(* IEC 61131-3 sources: SRCI/RobotLibrary/RobotLibrary/POUs/_internal, 7 files *)

(* ---- ActiveCommandRegisterFB.st ---- *)
FUNCTION_BLOCK ActiveCommandRegisterFB EXTENDS RobotLibraryLogFB
// -------------------------------------------------------------------------
//  SRCI Robot Library
// -------------------------------------------------------------------------
//
//  Object:      ActiveCommandRegisterFB
//  Author:      Thorsten Brach
//  Date:        2024-06-01
//
//  Description:
//
//
//  Copyright:
//    (C) 2024 Thorsten Brach. All rights reserved
//             Licensed under the LGPL-3.0 license.
//
//  Disclaimer:
//    This project is provided without any guarantee and can be used for
//    private and commercial purposes. Any use is at the user’s
//    own risk and responsibility.
//
// -------------------------------------------------------------------------
VAR_INPUT
  /// Active Command Register
  Register            : ARRAY [1..RobotLibraryParameter.ACTIVE_CMD_REGISTER_ENTRIES_MAX] OF AxesGroupAcyclicAcrEntry;
  /// System Time
  SystemTime          : DT;
END_VAR

VAR_OUTPUT
  /// Size of the register
  Size                : UINT := DINT_TO_UINT(RobotLibraryParameter.ACTIVE_CMD_REGISTER_ENTRIES_MAX);
  /// Execution Order List
  ExecutionOrderList  : ARRAY [1..RobotLibraryParameter.ACTIVE_CMD_REGISTER_ENTRIES_MAX] OF DINT;
END_VAR

VAR
  /// temporarty Active Command Register
  TmpRegister        : ARRAY [1..RobotLibraryParameter.ACTIVE_CMD_REGISTER_ENTRIES_MAX] OF AxesGroupAcyclicAcrEntry;
  /// last used unique ID
  LastUniqueID       : UINT;
  ///

END_VAR

VAR CONSTANT
  /// Active command
  ACTIVE_CMD           : UDINT := 1;
  /// Buffered command
  BUFFER_CMD           : UDINT := 2;
  /// Empty ARC entry
  EMPTY_ARC_ENTRY      : AxesGroupAcyclicAcrEntry;
  /// Empty command entry
  EMPTY_CMD_ENTRY      : AxesGroupAcyclicAcrEntryCmdBuffer;

  /// constant for byte index of priority in payload
  PRIORITY_IDX         : BYTE := 3;  /// bitmask to mask the priority out of the halfbyte
  PRIORITY_BIT_MASK    : BYTE := 2#000_1111;
END_VAR

  ManageRegister();

  UpdateExecutionOrderList();

END_FUNCTION_BLOCK

METHOD PUBLIC AddCmd : UDINT
VAR_INPUT
  /// Pointer to the corresponding command-FB to enable a callback mechanism
  pCommandFB   : POINTER TO RobotLibraryBaseFB;
END_VAR

VAR
  /// internal index for loops
 _regIdx     : DINT;
  /// internal command type
 _cmdType    : CmdType;
  /// log message
 _messageLog         : AlarmMessage;
END_VAR

  FOR _regIdx := 1 TO RobotLibraryParameter.ACTIVE_CMD_REGISTER_ENTRIES_MAX
  DO
    IF ( Register[_regIdx].State = ActiveCommandRegisterState.IS_FREE )
    THEN
      Register[_regIdx].State                        := ActiveCommandRegisterState.IS_PROCESSING;
      Register[_regIdx].UniqueID                     := CreateUniqueID();
      Register[_regIdx].pCommandFB                   := pCommandFB;

      // check pointer to command FB
      IF ( Register[_regIdx].pCommandFB <> RobotLibraryConstants.XNULL )
      THEN
        Register[_regIdx].Command[RobotLibraryConstants.ACTIVE_CMD].Timestamp  := SystemTime;
        Register[_regIdx].Command[RobotLibraryConstants.ACTIVE_CMD].Payload    := pCommandFB^.CommandData.Payload;
        Register[_regIdx].Command[RobotLibraryConstants.ACTIVE_CMD].PayloadLen := pCommandFB^.CommandData.PayloadLen;
        Register[_regIdx].Command[RobotLibraryConstants.ACTIVE_CMD].PayLoadPtr := 0;
        Register[_regIdx].Command[RobotLibraryConstants.ACTIVE_CMD].State      := BufferStateCmd.CREATED;
  		END_IF

      // return Unique ID
      AddCmd := Register[_regIdx].UniqueID;

      // Get CmdType from payload
      MemCpy( destAddr := ADR(_cmdType), ADR(pCommandFB^.CommandData.Payload), SIZEOF(_cmdType));

      // Create log entry
      CreateLogMessagePara1 ( Timestamp   := SystemTime,
                              MessageType := MessageType.CMD,
                              Severity    := Severity.DEBUG,
                              MessageCode := 0,
                              MessageText := 'Added Cmd <{1}> to active command register',
                              Para1       :=  CmdTypeToString(SwapUint(_cmdType)));
      EXIT;
  	END_IF
  END_FOR

END_METHOD

METHOD AddRsp : UDINT
VAR_INPUT
  /// Response
  Rsp : TelegramRobToPlcFragment;
END_VAR
VAR
  /// internal index for loops
 _Idx             : DINT;
  /// internal registen index
 _regIdx          : DINT;
  /// internal FragmentAction
 _fragmentAction  :  FragmentAction;
  /// internal command message state
 _cmdMessageState : CmdMessageState;
END_VAR

  FOR _regIdx := 1 TO RobotLibraryParameter.ACTIVE_CMD_REGISTER_ENTRIES_MAX
  DO
    IF ( Register[_regIdx].UniqueID = Rsp.Header.CmdID )
    THEN
      // convert to fragment action
     _fragmentAction := ByteToFragmentAction(Rsp.Header.FragmentAction);

      // delete response
      IF ( _fragmentAction.Clear )
      THEN
        MemSet( ADR(Register[_regIdx].Response[1]), 0, SIZEOF(Register[_regIdx].Response[1]));
      END_IF

      // add payload to response
      FOR _idx := Rsp.Header.PayloadPointer TO  Rsp.Header.PayloadLength -1
      DO
        Register[_regIdx].Response[1].Timestamp     := SystemTime;
        Register[_regIdx].Response[1].State         := BufferStateRsp.RECEIVING;
        Register[_regIdx].Response[1].PayloadLen    := Register[_regIdx].Response[1].PayloadLen + 1;
        Register[_regIdx].Response[1].Payload[_idx] := Rsp.Command.Payload[_idx];
      END_FOR

      // Get current message state
     _cmdMessageState := GetHalfeByteLo(Register[_regIdx].Response[1].Payload[0]);

      // Create log entry
      CreateLogMessagePara2 ( Timestamp   := SystemTime,
                              MessageType := MessageType.CMD,
                              Severity    := Severity.DEBUG,
                              MessageCode := 0,
                              MessageText := 'Added Rsp <{1}> with State = {2} to ACR',
                              Para1       :=  UINT_TO_STRING(Rsp.Header.CmdID),
                              Para2       :=  CmdMessageStateToString(_cmdMessageState));

      IF ( _fragmentAction.Complete )
      THEN
        // set response state
        Register[_regIdx].Response[1].State := BufferStateRsp.RECEIVED;

        // Check current message state and tag the register state as IS_FINAL, if needed
        IF ( _cmdMessageState >= CmdMessageState.DONE)
        THEN
          Register[_regIdx].State := ActiveCommandRegisterState.IS_FINAL;

          // Create log entry
          CreateLogMessagePara1( Timestamp   := SystemTime,
                                 MessageType := MessageType.CMD,
                                 Severity    := Severity.DEBUG,
                                 MessageCode := 0,
                                 MessageText := 'ARC Register for Rsp <{1}> has reached Final State',
                                 Para1       :=  UINT_TO_STRING(Rsp.Header.CmdID));
          // Exit the loop
  		  END_IF
      END_IF

      EXIT;
    END_IF
  END_FOR

END_METHOD

METHOD PRIVATE CreateUniqueID : UINT
VAR_INPUT
END_VAR

  // inc last unique ID
  LastUniqueID := LastUniqueID + 1;
  // return unique ID
  CreateUniqueID := LastUniqueID;

END_METHOD

METHOD FB_init : BOOL
VAR_INPUT
	bInitRetains : BOOL; // if TRUE, the retain variables are initialized (warm start / cold start)
	bInCopyCode : BOOL;  // if TRUE, the instance afterwards gets moved into the copy code (online change)
END_VAR

  MyType := 'ActiveCommandRegisterFB';

END_METHOD

METHOD PRIVATE ManageRegister
VAR
  /// internal index
 _regIdx     : DINT;
END_VAR

  FOR _regIdx := 1 TO RobotLibraryParameter.ACTIVE_CMD_REGISTER_ENTRIES_MAX
  DO
    // Check pointer to command FB is valid ?
    IF ( Register[_regIdx].pCommandFB = RobotLibraryConstants.XNULL)
    THEN
      RETURN;
  	END_IF

    // Check apply Cmd parameter update ?
    IF (( Register[_regIdx].Command[ACTIVE_CMD].State = BufferStateCmd.PROCESSED        ) AND
        ( Register[_regIdx].Command[BUFFER_CMD].State = BufferStateCmd.UPDATE_AVAILABLE ))
    THEN
      Register[_regIdx].Command[ACTIVE_CMD] := Register[_regIdx].Command[BUFFER_CMD];
      Register[_regIdx].Command[BUFFER_CMD] := EMPTY_CMD_ENTRY;
  	END_IF

    // Check Response received ?
    IF ( Register[_regIdx].Response[ACTIVE_CMD].State = BufferStateRsp.RECEIVED)
    THEN
      // update state
      Register[_regIdx].Response[ACTIVE_CMD].State := BufferStateRsp.PROCESSED;
      // callback CommandFB
      Register[_regIdx].pCommandFB^.CallBack(Register[_regIdx].Response[ACTIVE_CMD]);
  	END_IF

    // delete entries with State.IS_Final
    IF ( Register[_regIdx].State = ActiveCommandRegisterState.IS_FINAL )
    THEN
      // Create log entry
      CreateLogMessagePara2( Timestamp   := SystemTime,
                             MessageType := MessageType.CMD,
                             Severity    := Severity.DEBUG,
                             MessageCode := 0,
                             MessageText := 'Deleted ID <{1}> from ARC Register Idx <{2}> because of Final State was reached',
                             Para1       :=  UINT_TO_STRING(Register[_regIdx].UniqueID),
                             Para2       :=  DINT_TO_STRING(_regIdx) );

      Register[_regIdx] := EMPTY_ARC_ENTRY;
  	END_IF

  END_FOR

END_METHOD

PROPERTY PUBLIC NotifyParameterChanged : UDINT

SET
VAR
  /// internal register index
 _regIdx : DINT;
END_VAR

  FOR _regIdx := 1 TO RobotLibraryParameter.ACTIVE_CMD_REGISTER_ENTRIES_MAX
  DO
    // check unique ID found ?
    IF ( Register[_regIdx].UniqueID = NotifyParameterChanged )
    THEN
      IF (( Register[_regIdx].Command[ACTIVE_CMD].State <> BufferStateCmd.SENDING   ) AND
          ( Register[_regIdx].Command[ACTIVE_CMD].State <> BufferStateCmd.PROCESSED ))
      THEN
        // Check pointer is valid ?
        IF ( Register[_regIdx].pCommandFB <> RobotLibraryConstants.XNULL )
        THEN
          // add to send register
          Register[_regIdx].Command[ACTIVE_CMD].Timestamp  := SystemTime;
          Register[_regIdx].Command[ACTIVE_CMD].State      := BufferStateCmd.UPDATE_AVAILABLE;
          Register[_regIdx].Command[ACTIVE_CMD].Payload    := Register[_regIdx].pCommandFB^.CommandData.Payload;
          Register[_regIdx].Command[ACTIVE_CMD].PayloadLen := Register[_regIdx].pCommandFB^.CommandData.PayloadLen;

          // Create log entry
          CreateLogMessagePara2 ( Timestamp   := SystemTime,
                                  MessageType := MessageType.CMD,
                                  Severity    := Severity.DEBUG,
                                  MessageCode := 0,
                                  MessageText := 'Parameter update from {1} with CmdID <{2}> received -> written to ACTIVE_CMD Index',
                                  Para1       :=  Register[_regIdx].pCommandFB^.MyType,
                                  Para2       :=  UDINT_TO_STRING(NotifyParameterChanged));
  			END_IF
      ELSE
        // Check pointer is valid ?
        IF ( Register[_regIdx].pCommandFB <> RobotLibraryConstants.XNULL )
        THEN
          // add to buffer register
          Register[_regIdx].Command[BUFFER_CMD].Timestamp  := SystemTime;
          Register[_regIdx].Command[BUFFER_CMD].State      := BufferStateCmd.UPDATE_AVAILABLE;
          Register[_regIdx].Command[BUFFER_CMD].Payload    := Register[_regIdx].pCommandFB^.CommandData.Payload;
          Register[_regIdx].Command[BUFFER_CMD].PayloadLen := Register[_regIdx].pCommandFB^.CommandData.PayloadLen;

          // Create log entry
          CreateLogMessagePara2 ( Timestamp   := SystemTime,
                                  MessageType := MessageType.CMD,
                                  Severity    := Severity.DEBUG,
                                  MessageCode := 0,
                                  MessageText := 'Parameter update from {1} with CmdID <{2}> received -> written to BUFFER_CMD Index',
                                  Para1       :=  Register[_regIdx].pCommandFB^.MyType,
                                  Para2       :=  UDINT_TO_STRING(NotifyParameterChanged));
    		END_IF
  		END_IF

    END_IF
  END_FOR

END_SET

METHOD PUBLIC OnOnlineChange : DINT
VAR_INPUT
  /// unique ID
  UniqueID     : UDINT;
  /// Pointer to the corresponding command-FB to enable a callback mechanism
  pCommandFB   : POINTER TO RobotLibraryBaseFB;
END_VAR

VAR
  /// internal index for loops
 _regIdx : DINT;
END_VAR

  OnOnlineChange := -1;

  // Check command FB pointer is valid ?
  IF ( pCommandFB <> RobotLibraryConstants.XNULL)
  THEN
    FOR _regIdx := 1 TO RobotLibraryParameter.ACTIVE_CMD_REGISTER_ENTRIES_MAX
    DO
      // check unique ID found ?
      IF ( Register[_regIdx].UniqueID = UniqueID )
      THEN
        // update pointer to command FB
        Register[_regIdx].pCommandFB := pCommandFB;
        // Return result OK
        OnOnlineChange := RobotLibraryConstants.OK;
        EXIT;
      END_IF
    END_FOR
  END_IF

END_METHOD

METHOD PUBLIC RemoveCmd
VAR_INPUT
 /// unique ID
 UniqueID : UDINT;
END_VAR

VAR
  /// internal index
 _regIdx : DINT;
END_VAR

  FOR _regIdx := 1 TO RobotLibraryParameter.ACTIVE_CMD_REGISTER_ENTRIES_MAX
  DO
    // check unique ID found and not yet sended ?
    IF (( Register[_regIdx].UniqueID         = UniqueID               ) AND
        ( Register[_regIdx].Command[1].State < BufferStateCmd.SENDING ))
    THEN
      // delete register entry
      MemSet(ADR(Register[_regIdx]), 0 , SIZEOF(Register[_regIdx]));
      EXIT;
    END_IF
  END_FOR

END_METHOD

METHOD PRIVATE UpdateExecutionOrderList
VAR
  /// temporary Active Command Register entry
  TmpRegisterEntry : AxesGroupAcyclicAcrEntry;
  /// temporary index
  TmpIndex         : DINT;
  /// internal index
  i                : DINT;
  /// internal index
  j                : DINT;
END_VAR

  // Reset temporary register
  MemSet(destAddr := ADR(TmpRegister)       , fillByte := 0, n := SIZEOF(TmpRegister));
  // Reset Execution Order List
  MemSet(destAddr := ADR(ExecutionOrderList), fillByte := 0, n := SIZEOF(ExecutionOrderList));
  // pre-set temporary register index
  j := 1;

  FOR i := 1 TO RobotLibraryParameter.ACTIVE_CMD_REGISTER_ENTRIES_MAX
  DO
    // add only entries which are not in status free
    IF ( Register[i].State >  ActiveCommandRegisterState.IS_FREE )
    THEN
      // copy register entry
      TmpRegister[j] := Register[i];
      // store index of the entry from the ARC
      ExecutionOrderList[j] := i;
      // inc temporar register index
      j := j + 1;
  	END_IF
  END_FOR

  // Bubble Sort to sort the priorities from the active command register
  FOR i := 1 TO RobotLibraryParameter.ACTIVE_CMD_REGISTER_ENTRIES_MAX
  DO
    FOR j := 1 TO RobotLibraryParameter.ACTIVE_CMD_REGISTER_ENTRIES_MAX - 1
    DO
      // check list entry is not empty ?
      IF (( TmpRegister[i  ].State = ActiveCommandRegisterState.IS_FREE ) OR
          ( TmpRegister[j+1].State = ActiveCommandRegisterState.IS_FREE ))
      THEN
        EXIT;
      END_IF

      IF (( TmpRegister[j].Command[ACTIVE_CMD].Payload[PRIORITY_IDX] AND PRIORITY_BIT_MASK ) > ( TmpRegister[j+1].Command[ACTIVE_CMD].Payload[PRIORITY_IDX] AND PRIORITY_BIT_MASK ))
      THEN
        // swap position of register entry
        TmpRegisterEntry := TmpRegister[j];
        TmpRegister[j]   := TmpRegister[j+1];
        TmpRegister[j+1] := TmpRegisterEntry;

        // swap position of index in the Execution Order List
        TmpIndex                := ExecutionOrderList[j];
        ExecutionOrderList[j]   := ExecutionOrderList[j+1];
        ExecutionOrderList[j+1] := TmpIndex;
      END_IF
    END_FOR
  END_FOR

  // Bubble Sort to sort the Timestamp from the pre-sorted active command register
  FOR i := 1 TO RobotLibraryParameter.ACTIVE_CMD_REGISTER_ENTRIES_MAX
  DO
    FOR j := 1 TO RobotLibraryParameter.ACTIVE_CMD_REGISTER_ENTRIES_MAX - 1
    DO
      // check list entry is not empty ?
      IF (( TmpRegister[i  ].State = ActiveCommandRegisterState.IS_FREE ) OR
          ( TmpRegister[j+1].State = ActiveCommandRegisterState.IS_FREE ))
      THEN
        EXIT;
      END_IF

      IF (( TmpRegister[j].Command[ACTIVE_CMD].Payload[PRIORITY_IDX] AND PRIORITY_BIT_MASK ) >= ( TmpRegister[j+1].Command[ACTIVE_CMD].Payload[PRIORITY_IDX] AND PRIORITY_BIT_MASK )) AND
         (( TmpRegister[j].Command[ACTIVE_CMD].Timestamp )                                   >  ( TmpRegister[j+1].Command[ACTIVE_CMD].Timestamp ))
      THEN
        // swap position of register entry
        TmpRegisterEntry := TmpRegister[j];
        TmpRegister[j]   := TmpRegister[j+1];
        TmpRegister[j+1] := TmpRegisterEntry;

        // swap position of index in the Execution Order List
        TmpIndex                := ExecutionOrderList[j];
        ExecutionOrderList[j]   := ExecutionOrderList[j+1];
        ExecutionOrderList[j+1] := TmpIndex;
      END_IF
    END_FOR
  END_FOR

END_METHOD

(* ---- RecvData.st ---- *)
{attribute 'pack_mode' := '1'}
FUNCTION_BLOCK RecvData
// -------------------------------------------------------------------------
//  SRCI Robot Library
// -------------------------------------------------------------------------
//
//  Object:      RecvData
//  Author:      Thorsten Brach
//  Date:        2024-06-01
//
//  Description:
//
//
//  Copyright:
//    (C) 2024 Thorsten Brach. All rights reserved
//             Licensed under the LGPL-3.0 license.
//
//  Disclaimer:
//    This project is provided without any guarantee and can be used for
//    private and commercial purposes. Any use is at the user’s
//    own risk and responsibility.
//
// -------------------------------------------------------------------------
VAR_INPUT
  /// Payload
  Payload    : ARRAY [0..RobotLibraryParameter.TELEGRAM_PAYLOAD_MAX] OF BYTE;
  /// Payload length
  PayloadLen : UDINT;
  /// Payload pointer
  PayloadPtr : DINT;
END_VAR

END_FUNCTION_BLOCK

/// returns a ArmConfigParameter from the payload buffer from the current payload pointer address and increase the payload pointer afterwards
METHOD GetArmConfig : ArmConfigParameter
VAR
  /// temporary byte
 _tmpByte : BYTE;
END_VAR

  // get 1st Byte
  _tmpByte := GetByte();

  GetArmConfig.Shoulder.0 := _tmpByte.0;
  GetArmConfig.Elbow.0    := _tmpByte.1;
  GetArmConfig.Wrist.0    := _tmpByte.2;

  // get 2nd byte to inc the PayloadPointer
  _tmpByte := GetByte();

END_METHOD

/// returns a BOOL from the payload buffer from the current payload pointer address and increase the payload pointer afterwards
METHOD GetBool : BOOL

  // copy data
  GetBool := Payload[PayloadPtr].0;
  // inc payload pointer
  PayloadPtr := PayloadPtr + SIZEOF(BYTE);

END_METHOD

/// returns a BYTE from the payload buffer from the current payload pointer address and increase the payload pointer afterwards
METHOD GetByte : BYTE

  // copy data
  GetByte := Payload[PayloadPtr];
  // inc payload pointer
  PayloadPtr := PayloadPtr + SIZEOF(BYTE);

END_METHOD

/// returns a datablock from the payload buffer from the current payload pointer address and increase the payload pointer afterwards
METHOD GetDataBlock
VAR_INPUT
  /// Target
  pData    : POINTER TO BYTE;
  /// Size of data block
  Size     : UDINT;
  /// Target data type is string ?
  IsString : BOOL;
END_VAR

  IF ( pData <> RobotLibraryConstants.XNULL)
  THEN
    IF ( IsString)
    THEN
      Size := Size -1;
  	END_IF

    // copy data
    MemCpy(pData, ADR(Payload[PayloadPtr]), Size);

    // inc payload pointer
    PayloadPtr := PayloadPtr + UDINT_TO_DINT(Size);
  END_IF

END_METHOD

/// returns a DataInSync from the payload buffer from the current payload pointer address and increase the payload pointer afterwards
METHOD GetDataInSync : DataInSync
VAR
  /// temporary byte
 _tmpByte : BYTE;
END_VAR

  // copy data
  _tmpByte := Payload[PayloadPtr];

  GetDataInSync.ToolsInSync             := _tmpByte.0;
  GetDataInSync.FramesInSync            := _tmpByte.1;
  GetDataInSync.LoadsInSync             := _tmpByte.2;
  GetDataInSync.WorkAreasInSync         := _tmpByte.3;
  GetDataInSync.SoftwareLimitsInSync    := _tmpByte.4;
  GetDataInSync.DefaultDynamicsInSync   := _tmpByte.5;
  GetDataInSync.ReferenceDynamicsInSync := _tmpByte.6;

  // inc payload pointer
  PayloadPtr := PayloadPtr + SIZEOF(BYTE);

END_METHOD

/// returns a DWORD from the payload buffer from the current payload pointer address and increase the payload pointer afterwards
METHOD GetDword : DWORD

  // copy data
  MemCpy(ADR(GetDword), ADR(Payload[PayloadPtr]), SIZEOF(DWORD));
  // inc payload pointer
  PayloadPtr := PayloadPtr + SIZEOF(DWORD);

END_METHOD

/// returns a FragmentAction from the payload buffer from the current payload pointer address and increase the payload pointer afterwards
METHOD GetFragmentAction : FragmentAction
VAR
  /// temporary byte
 _tmpByte : BYTE;
END_VAR

  // copy data
  _tmpByte := Payload[PayloadPtr];

  GetFragmentAction.Complete := _tmpByte.0;
  GetFragmentAction.Reset    := _tmpByte.1;
  GetFragmentAction.Clear    := _tmpByte.2;
  GetFragmentAction.BIT03    := _tmpByte.3;
  GetFragmentAction.BIT04    := _tmpByte.4;
  GetFragmentAction.BIT05    := _tmpByte.5;
  GetFragmentAction.BIT06    := _tmpByte.6;
  GetFragmentAction.BIT07    := _tmpByte.7;

  // inc payload pointer
  PayloadPtr := PayloadPtr + SIZEOF(BYTE);

END_METHOD

/// returns the 1st halfe BYTE from the payload buffer from the current payload pointer address and increase the payload pointer afterwards
METHOD GetHalfeByte1 : BYTE
VAR_INPUT
  /// Increase payload pointer
  IncPayloadPtr : BOOL;
END_VAR

VAR
  /// temporary byte
 _tmpByte : BYTE;
END_VAR

  // copy data
  _tmpByte := Payload[PayloadPtr];

  GetHalfeByte1.0 := _tmpByte.0;
  GetHalfeByte1.1 := _tmpByte.1;
  GetHalfeByte1.2 := _tmpByte.2;
  GetHalfeByte1.3 := _tmpByte.3;

  IF (IncPayloadPtr)
  THEN
    // inc payload pointer
    PayloadPtr := PayloadPtr + SIZEOF(BYTE);
  END_IF

END_METHOD

/// returns the 1st halfe BYTE from the payload buffer from the current payload pointer address and increase the payload pointer afterwards
METHOD GetHalfeByte2 : BYTE
VAR_INPUT
  /// Increase payload pointer
  IncPayloadPtr : BOOL;
END_VAR

VAR
  /// temporary byte
 _tmpByte : BYTE;
END_VAR

  // copy data
  _tmpByte := Payload[PayloadPtr];

  GetHalfeByte2.0 := _tmpByte.4;
  GetHalfeByte2.1 := _tmpByte.5;
  GetHalfeByte2.2 := _tmpByte.6;
  GetHalfeByte2.3 := _tmpByte.7;

  IF (IncPayloadPtr)
  THEN
    // inc payload pointer
    PayloadPtr := PayloadPtr + SIZEOF(BYTE);
  END_IF

END_METHOD

/// returns a IEC_Date from the payload buffer from the current payload pointer address and increase the payload pointer afterwards
METHOD GetIecDate : IEC_Date

  // copy data
  MemCpy(ADR(GetIecDate), ADR(Payload[PayloadPtr]), SIZEOF(IEC_DATE));
  // swap byte order
  GetIecDate := SwapIecDate(GetIecDate);
  // inc payload pointer
  PayloadPtr := PayloadPtr + SIZEOF(IEC_DATE);

END_METHOD

/// returns a IEC_TIME from the payload buffer from the current payload pointer address and increase the payload pointer afterwards
METHOD GetIecTime : IEC_TIME

  // copy data
  MemCpy(ADR(GetIecTime), ADR(Payload[PayloadPtr]), SIZEOF(IEC_TIME));
  // swap byte order
  GetIecTime := SwapIecTime(GetIecTime);
  // inc payload pointer
  PayloadPtr := PayloadPtr + SIZEOF(IEC_TIME);

END_METHOD

/// returns a INT from the payload buffer from the current payload pointer address and increase the payload pointer afterwards
METHOD GetInt : INT

  // copy data
  MemCpy(ADR(GetInt), ADR(Payload[PayloadPtr]), SIZEOF(INT));
  // swap byte order
  GetInt := SwapInt(GetInt);
  // inc payload pointer
  PayloadPtr := PayloadPtr + SIZEOF(INT);

END_METHOD

/// returns a REAL from the payload buffer from the current payload pointer address and increase the payload pointer afterwards
METHOD GetReal : REAL

  // copy data
  MemCpy(ADR(GetReal), ADR(Payload[PayloadPtr]), SIZEOF(REAL));
  // swap byte order
  GetReal := SwapReal(GetReal);
  // inc payload pointer
  PayloadPtr := PayloadPtr + SIZEOF(Real);

END_METHOD

/// returns a SINT from the payload buffer from the current payload pointer address and increase the payload pointer afterwards
METHOD GetSint : SINT

  // copy data
  MemCpy(ADR(GetSint), ADR(Payload[PayloadPtr]), SIZEOF(SINT));
  // inc payload pointer
  PayloadPtr := PayloadPtr + SIZEOF(SINT);

END_METHOD

/// returns a String from the payload buffer from the current payload pointer address and increase the payload pointer afterwards
METHOD GetString : STRING(255)
VAR_INPUT
  Size : DINT;
END_VAR

  // copy data
  MemCpy(ADR(GetString), ADR(Payload[PayloadPtr]), DINT_TO_UDINT(Size));

  // inc payload pointer
  PayloadPtr := PayloadPtr + Size;

END_METHOD

/// returns a TrackingStatus from the payload buffer from the current payload pointer address and increase the payload pointer afterwards
METHOD GetTrackingStatus : TrackingStatus
VAR
  /// temporary byte
  tmpByte : BYTE;
END_VAR

  // copy data
  tmpByte := GetByte();

  GetTrackingStatus.ConveyorTrackingEnabled   := tmpByte.0;
  GetTrackingStatus.WaitingForSynchronization := tmpByte.1;
  GetTrackingStatus.Synchronizing             := tmpByte.2;
  GetTrackingStatus.Synchronous               := tmpByte.3;
  GetTrackingStatus.Desynchronizing           := tmpByte.4;
  GetTrackingStatus.SyncOutZoneEntered        := tmpByte.5;
  GetTrackingStatus.SyncOutZoneLeft           := tmpByte.6;
  GetTrackingStatus.NotUsed                   := tmpByte.7;

END_METHOD

/// returns a TurnNumber from the payload buffer from the current payload pointer address and increase the payload pointer afterwards
METHOD GetTurnNumbers : TurnNumber

  GetTurnNumbers.J1Turns := BYTE_TO_SINT(GetHalfeByte1(FALSE));
  GetTurnNumbers.J2Turns := BYTE_TO_SINT(GetHalfeByte2(TRUE));

  GetTurnNumbers.J3Turns := BYTE_TO_SINT(GetHalfeByte1(FALSE));
  GetTurnNumbers.J4Turns := BYTE_TO_SINT(GetHalfeByte2(TRUE));

  GetTurnNumbers.J5Turns := BYTE_TO_SINT(GetHalfeByte1(FALSE));
  GetTurnNumbers.J6Turns := BYTE_TO_SINT(GetHalfeByte2(TRUE));

  GetTurnNumbers.E1Turns := BYTE_TO_SINT(GetByte());

END_METHOD

/// returns a UDINT from the payload buffer from the current payload pointer address and increase the payload pointer afterwards
METHOD GetUdint : UDINT

  // copy data
  MemCpy(ADR(GetUdint), ADR(Payload[PayloadPtr]), SIZEOF(UDINT));
  // swap byte order
  GetUdint := SwapUdint(GetUdint);
  // inc payload pointer
  PayloadPtr := PayloadPtr + SIZEOF(UDINT);

END_METHOD

/// returns a UINT from the payload buffer from the current payload pointer address and increase the payload pointer afterwards
METHOD GetUint : UINT

  // copy data
  MemCpy(ADR(GetUint), ADR(Payload[PayloadPtr]), SIZEOF(UINT));
  // swap byte order
  GetUint := SwapUint(GetUint);
  // inc payload pointer
  PayloadPtr := PayloadPtr + SIZEOF(UINT);

END_METHOD

/// returns a USINT from the payload buffer from the current payload pointer address and increase the payload pointer afterwards
METHOD GetUsint : USINT

  // copy data
  MemCpy(ADR(GetUsint), ADR(Payload[PayloadPtr]), SIZEOF(USINT));
  // inc payload pointer
  PayloadPtr := PayloadPtr + SIZEOF(USINT);

END_METHOD

/// returns a WORD from the payload buffer from the current payload pointer address and increase the payload pointer afterwards
METHOD GetWord : WORD

  // copy data
  MemCpy(ADR(GetWord), ADR(Payload[PayloadPtr]), SIZEOF(WORD));
  // swap byte order
  GetWord := SwapWord(GetWord);
  // inc payload pointer
  PayloadPtr := PayloadPtr + SIZEOF(WORD);

END_METHOD

/// Resets the payload buffer, the payload pointer and the payload length
METHOD Reset
VAR_INPUT
END_VAR

  MemSet(ADR(Payload), 0 , SIZEOF(Payload));
  PayloadLen := 0;
  PayloadPtr := 0;

END_METHOD

(* ---- RobotLibraryBaseEnableFB.st ---- *)
FUNCTION_BLOCK RobotLibraryBaseEnableFB EXTENDS RobotLibraryBaseFB
// -------------------------------------------------------------------------
//  SRCI Robot Library
// -------------------------------------------------------------------------
//
//  Object:      RobotLibraryBaseFB
//  Author:      Thorsten Brach
//  Date:        2024-08-11
//
//  Description:
//
//
//  Copyright:
//    (C) 2024 Thorsten Brach. All rights reserved
//             Licensed under the LGPL-3.0 license.
//
//  Disclaimer:
//    This project is provided without any guarantee and can be used for
//    private and commercial purposes. Any use is at the user’s
//    own risk and responsibility.
//
// -------------------------------------------------------------------------
VAR_INPUT
  /// Set TRUE to activate / Set False to deactivate
  Enable            : BOOL;
END_VAR

VAR_OUTPUT
  /// FB is being processed
  Busy              : BOOL;
  /// Command is transferred and confirmed by the RC
//CommandBuffered   : BOOL;
  /// TRUE while function is active
  Enabled           : BOOL;
  /// Receiving of input parameter values has been acknowledged by RC
//ParameterAccepted : BOOL;
END_VAR

VAR
  /// step counter for finite state machine
 _fsmState          : FsmState;
  /// Rising edge for enable
 _enable_R          : R_TRIG;
  /// Falling edge for enable
 _enable_F          : F_TRIG;
END_VAR

  SUPER^(AxesGroup := AxesGroup);

END_FUNCTION_BLOCK

METHOD internal FSM : DINT
VAR
  /// internal return value
 _retVal : DINT;
END_VAR

  CASE _fsmState
  OF

    FsmState.READY :

      // Await start
      IF (( NOT Busy       ) AND
          ( NOT Error      ) AND
          (    _enable_R.Q ))
      THEN
        // inc fsm step
       _fsmState := FsmState.START;
  	  END_IF

    FsmState.START :

     _retVal := OnExecStart();

      IF ( _retVal = RobotLibraryConstants.OK )
      THEN
       _fsmState := FsmState.RUNNING;
      ELSE
        // Cancel
        IF ((      Busy       ) AND
            (  NOT Error      ) AND
            (     _enable_F.Q ))
        THEN
         _fsmState := FsmState.CANCEL;
          RETURN;
  			END_IF

        // check error
        IF (_retVal < RobotLibraryConstants.OK)
        THEN
         _fsmState := FsmState.ERROR;
          RETURN;
  			END_IF
  		END_IF

     FsmState.RUNNING :

        _retVal := OnExecRun();

         IF (_retVal = RobotLibraryConstants.OK )
         THEN
          _fsmState := FsmState.DONE;
         ELSE
           // Cancel
           IF ((      Busy       ) AND
               (  NOT Error      ) AND
               (     _enable_F.Q ))
           THEN
            _fsmState := FsmState.CANCEL;
             RETURN;
  				 END_IF

           // error
           IF (_retVal < RobotLibraryConstants.OK)
           THEN
            _fsmState := 99;
             RETURN;
  				 END_IF
  			 END_IF

    FsmState.DONE :

     _fsmState := FsmState.READY;

    FsmState.CANCEL :

     _retVal := OnExecCancel();

      IF (_retVal = RobotLibraryConstants.OK )
      THEN
        _fsmState := FsmState.READY;
      END_IF

    FsmState.ERROR :

      IF (NOT Enable)
      THEN
       _fsmState := FsmState.ERROR_CLEAR;
  		END_IF

    FsmState.ERROR_CLEAR :

     _retVal := OnExecErrorClear();

      IF (_retVal = RobotLibraryConstants.OK )
      THEN
        _fsmState := FsmState.READY;
      END_IF

  ELSE
    ;
  END_CASE

END_METHOD

METHOD PROTECTED OnCall
VAR_IN_OUT
  /// Robot assignment of function
  AxesGroup         : AxesGroup;
END_VAR

  SUPER^.OnCall(AxesGroup := AxesGroup);

  // building rising and falling edges
  _enable_R( CLK := Enable);
  _enable_F( CLK := Enable);

  // call state machine
  FSM();

END_METHOD

METHOD Protected OnExecCancel : DINT
VAR_INPUT
END_VAR

  OnExecCancel := Reset();

  // Create log entry
  CreateLogMessagePara1 ( Timestamp   := AxesGroup.InternalData.SystemTime,
                          MessageType := MessageType.CMD,
                          Severity    := Severity.DEBUG,
                          MessageCode := 0,
                          MessageText := 'Execution of FB {1} cancled ',
                          Para1       := MyType);

END_METHOD

METHOD PROTECTED OnExecErrorClear : DINT
VAR_INPUT
END_VAR

  Reset();

END_METHOD

METHOD PROTECTED OnExecRun : DINT
VAR_INPUT
END_VAR

END_METHOD

METHOD PROTECTED OnExecStart : DINT
VAR_INPUT
END_VAR

END_METHOD

METHOD PROTECTED Reset : DINT
VAR_INPUT
END_VAR

  Reset := SUPER^.Reset();

  Busy    := FALSE;
  Enabled := FALSE;

END_METHOD

(* ---- RobotLibraryBaseExecuteFB.st ---- *)
FUNCTION_BLOCK RobotLibraryBaseExecuteFB extends RobotLibraryBaseFB
// -------------------------------------------------------------------------
//  SRCI Robot Library
// -------------------------------------------------------------------------
//
//  Object:      RobotLibraryBaseFB
//  Author:      Thorsten Brach
//  Date:        2024-08-11
//
//  Description:
//
//
//  Copyright:
//    (C) 2024 Thorsten Brach. All rights reserved
//             Licensed under the LGPL-3.0 license.
//
//  Disclaimer:
//    This project is provided without any guarantee and can be used for
//    private and commercial purposes. Any use is at the user’s
//    own risk and responsibility.
//
// -------------------------------------------------------------------------
VAR_INPUT
  /// Start of the command at the rising edge
  Execute         : BOOL;
END_VAR
VAR_OUTPUT
  /// The command has been completed successfully
  Done            : BOOL;
  /// FB is being processed
  Busy            : BOOL;
  /// Command is transferred and confirmed by the RC
//  CommandBuffered : BOOL;
END_VAR

VAR
  /// step counter for finite state machine
 _fsmState        : FsmState;
  /// Rising edge for execute
 _execute_R       : R_TRIG;
  /// Falling edge for execute
 _execute_F       : F_TRIG;
END_VAR

  SUPER^(AxesGroup := AxesGroup);

END_FUNCTION_BLOCK

METHOD INTERNAL ApplyOutCmd
VAR_INPUT
END_VAR

END_METHOD

METHOD INTERNAL ApplyParCmd
VAR_INPUT
END_VAR

END_METHOD

METHOD internal FSM : DINT
VAR
  /// internal return value
 _retVal : DINT;
END_VAR

  CASE _fsmState
  OF

    FsmState.READY :

      // Await start
      IF (( NOT Busy        ) AND
          ( NOT Error       ) AND
          (    _execute_R.Q ))
      THEN
        // inc fsm step
       _fsmState := FsmState.START;
  	  END_IF

    FsmState.START :

     _retVal := OnExecStart();

      IF ( _retVal = RobotLibraryConstants.OK )
      THEN
       _fsmState := FsmState.RUNNING;
      ELSE
        // Cancel
        IF ((      Busy        ) AND
            (  NOT Error       ) AND
            (     _execute_F.Q ))
        THEN
         _fsmState := FsmState.CANCEL;
          RETURN;
  			END_IF

        // check error
        IF (_retVal < RobotLibraryConstants.OK)
        THEN
         _fsmState := FsmState.ERROR;
          RETURN;
  			END_IF
  		END_IF

     FsmState.RUNNING :

        _retVal := OnExecRun();

         IF (_retVal = RobotLibraryConstants.OK )
         THEN
          _fsmState := FsmState.DONE;
         ELSE
           // Cancel
           IF ((      Busy        ) AND
               (  NOT Error       ) AND
               (     _execute_F.Q ))
           THEN
            _fsmState := FsmState.CANCEL;
             RETURN;
  				 END_IF

           // error
           IF (_retVal < RobotLibraryConstants.OK)
           THEN
            _fsmState := 99;
             RETURN;
  				 END_IF
  			 END_IF

    FsmState.DONE :

     _fsmState := FsmState.READY;

    FsmState.CANCEL :

     _retVal := OnExecCancel();

      IF (_retVal = RobotLibraryConstants.OK )
      THEN
        _fsmState := FsmState.READY;
      END_IF

    FsmState.ERROR :

      IF (NOT Execute)
      THEN
       _fsmState := FsmState.ERROR_CLEAR;
  		END_IF

    FsmState.ERROR_CLEAR :

     _retVal := OnExecErrorClear();

      IF (_retVal = RobotLibraryConstants.OK )
      THEN
        _fsmState := FsmState.READY;
      END_IF

  ELSE
    ;
  END_CASE

END_METHOD

// Base implementation must be called !
METHOD PROTECTED OnCall
VAR_IN_OUT
  /// Robot assignment of function
  AxesGroup         : AxesGroup;
END_VAR

  SUPER^.OnCall(AxesGroup := AxesGroup);

  // building rising and falling edges
  _execute_R( CLK := Execute);
  _execute_F( CLK := EXecute);

  // call state machine
  FSM();

END_METHOD

METHOD PROTECTED OnExecCancel : DINT
VAR_INPUT
END_VAR

  OnExecCancel := Reset();

  // Create log entry
  CreateLogMessagePara1 ( Timestamp   := AxesGroup.InternalData.SystemTime,
                          MessageType := MessageType.CMD,
                          Severity    := Severity.DEBUG,
                          MessageCode := 0,
                          MessageText := 'Execution of FB {1} cancled ',
                          Para1       := MyType);

END_METHOD

METHOD PROTECTED OnExecErrorClear : DINT
VAR_INPUT
END_VAR

  Reset();

END_METHOD

METHOD PROTECTED OnExecRun : DINT
VAR_INPUT
END_VAR

END_METHOD

METHOD PROTECTED OnExecStart : DINT
VAR_INPUT
END_VAR

END_METHOD

METHOD PROTECTED Reset : DINT
VAR_INPUT
END_VAR

  Reset := SUPER^.Reset();

  Done := FALSE;
  Busy := FALSE;

END_METHOD

(* ---- RobotLibraryBaseFB.st ---- *)
FUNCTION_BLOCK RobotLibraryBaseFB EXTENDS RobotLibraryLogFB
// -------------------------------------------------------------------------
//  SRCI Robot Library
// -------------------------------------------------------------------------
//
//  Object:      RobotLibraryBaseFB
//  Author:      Thorsten Brach
//  Date:        2024-06-01
//
//  Description:
//
//
//  Copyright:
//    (C) 2024 Thorsten Brach. All rights reserved
//             Licensed under the LGPL-3.0 license.
//
//  Disclaimer:
//    This project is provided without any guarantee and can be used for
//    private and commercial purposes. Any use is at the user’s
//    own risk and responsibility.
//
// -------------------------------------------------------------------------
VAR_INPUT
  /// User defined command name
  Name         : STRING(20);
  /// Execution Mode
  ExecMode     : ExecutionMode;
  /// Priority
  Priority     : PriorityLevel;
END_VAR
VAR_OUTPUT
  /// Command data
  CommandData  : SendData;
  /// response data
  ResponseData : RecvData;
  /// An error occurred during the execution of the command
  Error        : BOOL;
  /// ErrorID reported by RC for error identification according to Table 7-1
  ErrorID      : WORD;
  ErrorIdEnum  : RobotLibraryErrorIdEnum;
  ErrorAddTxt  : STRING(RobotLibraryConstants.MAX_ADD_TEXT_LENGTH);

  /// WarningID for warning identification reported during execution of command according to Table 7-3
  WarningID    : WORD;
  WarningIdEnum: RobotLibraryWarningIdEnum;
  /// InfoID for info identification reported during execution of command according to Table 7-5
  InfoID       : WORD;
  InfoIdEnum   : RobotLibraryInfoIdEnum;
END_VAR
VAR_IN_OUT
  /// Robot assignment of function
  AxesGroup    : AxesGroup;
END_VAR

VAR
  /// Rising edge for error
 _error_R          : R_TRIG;
  /// Rising edge for warning
 _warning_R        : R_TRIG;
  /// Rising edge for information
 _info_R           : R_TRIG;
  /// unique ID
 _uniqueID         : UDINT;
  /// flag for response received
 _responseReceived : BOOL;
  /// internal step counter
 _stepCmd          : DINT;
  /// internal timer
 _timerCmd         : TON;
  /// internal timeout
 _timeoutCmd       : TIME := T#5S;
  /// internal command header
 _cmdHeader        : CmdHeader;
  /// internal response header
 _rspHeader        : RspHeader;
END_VAR

  OnCall               (AxesGroup := AxesGroup);
  CheckParameterChanged(AxesGroup := AxesGroup);

  IF ( AxesGroup.InternalData.OnlineChange_R.Q )
  THEN
    OnOnlineChange(AxesGroup := AxesGroup);
  END_IF

END_FUNCTION_BLOCK

METHOD PUBLIC CallBack : DINT
VAR_INPUT
  /// Response data
  RspData : AxesGroupAcyclicAcrEntryRspBuffer;
END_VAR

  ResponseData.Reset();
  ResponseData.Payload    := RspData.Payload;
  ResponseData.PayloadLen := RspData.PayloadLen;
  ParseResponsePayload(ResponseData);

  // set flag for response received
  _responseReceived := TRUE;

  // Create log entry
  CreateLogMessage ( Timestamp   := AxesGroup.InternalData.SystemTime,
                     MessageType := MessageType.CMD,
                     Severity    := Severity.DEBUG,
                     MessageCode := 0,
                     MessageText := CONCAT('Callback reveiced in FB ', MyType));

END_METHOD

METHOD CheckParameterChanged : BOOL
VAR_IN_OUT
  /// Robot assignment of function
  AxesGroup    : AxesGroup;
END_VAR

  IF ( CheckParameterChanged )
  THEN
    AxesGroup.Acyclic.ActiveCommandRegister.NotifyParameterChanged := _uniqueID;
  END_IF

END_METHOD

METHOD INTERNAL CreateCommandPayload : SendData

  // Reset all variables
  CreateCommandPayload.Reset();
  // Add CmdType
  CreateCommandPayload.AddUint(_cmdHeader.CmdTyp);
  // Add Reserve_ExecMode
  CreateCommandPayload.AddHalfBytes(  0               , _cmdHeader.ExecMode);
  // Add ParSeq_Priority
  CreateCommandPayload.AddHalfBytes( _cmdHeader.ParSeq, _cmdHeader.Priority);

END_METHOD

METHOD PROTECTED OnCall
VAR_IN_OUT
  /// Robot assignment of function
  AxesGroup         : AxesGroup;
END_VAR

  // map numeric value to enum, so that the corresponding message text is directly shown by the tooltip
  ErrorIdEnum   := ErrorId;
  WarningIdEnum := WarningId;
  InfoIdEnum    := InfoId;

  Error := ErrorID <> RobotLibraryConstants.OK;

  ExternalLogger := AxesGroup.MessageLog.ExternalLogger;
  LogLevel       := AxesGroup.MessageLog.LogLevel;

  // building rising edges for error, warning, info number detected
  _error_R  ( CLK := ErrorID   <> RobotLibraryConstants.OK );
  _warning_R( CLK := WarningID <> RobotLibraryConstants.OK );
  _info_R   ( CLK := InfoID    <> RobotLibraryConstants.OK );

  IF ( _error_R.Q)
  THEN
    // Create log entry
    CreateLogMessagePara2 ( Timestamp   := AxesGroup.InternalData.SystemTime,
                            MessageType := MessageType.CMD,
                            Severity    := Severity.DEBUG,
                            MessageCode := 0,
                            MessageText := 'Error with ID: 16#{1} in FB {2} received ',
                            Para1       := WORD_TO_STRING_HEX(ErrorID),
                            Para2       := MyType);
  END_IF

  IF ( _warning_R.Q)
  THEN
    // Create log entry
    CreateLogMessagePara2 ( Timestamp   := AxesGroup.InternalData.SystemTime,
                            MessageType := MessageType.CMD,
                            Severity    := Severity.DEBUG,
                            MessageCode := 0,
                            MessageText := 'Warning with ID: 16#{1} in FB {2} received ',
                            Para1       := WORD_TO_STRING_HEX(WarningID),
                            Para2       := MyType);
  END_IF

  IF ( _info_R.Q)
  THEN
    // Create log entry
    CreateLogMessagePara2 ( Timestamp   := AxesGroup.InternalData.SystemTime,
                            MessageType := MessageType.CMD,
                            Severity    := Severity.DEBUG,
                            MessageCode := 0,
                            MessageText := 'Info with ID: 16#{1} in FB {2} received ',
                            Para1       := WORD_TO_STRING_HEX(InfoID),
                            Para2       := MyType);
  END_IF

END_METHOD

METHOD OnOnlineChange : DINT
VAR_IN_OUT
  /// Robot assignment of function
  AxesGroup : AxesGroup;
END_VAR

  // update pointer to command FB
  AxesGroup.Acyclic.ActiveCommandRegister.OnOnlineChange( UniqueID := _uniqueID, pCommandFB := ADR(THIS^));

END_METHOD

METHOD INTERNAL ParseResponsePayload : DINT
VAR_INPUT
  /// Response data
  ResponseData : RecvData;
END_VAR

  // reset message IDs
  InfoID    := 0;
  WarningID := 0;
  ErrorID   := 0;

  // get State
  _rspHeader.State                := ResponseData.GetHalfeByte1(IncPayloadPtr := FALSE);
  // get ParSeq
  _rspHeader.ParSeq               := ResponseData.GetHalfeByte2(IncPayloadPtr := TRUE);
  // get AlarmMessageSeverity
  _rspHeader.AlarmMessageSeverity := ResponseData.GetByte();
  // get AlarmMessageCode
  _rspHeader.AlarmMessageCode     := ResponseData.GetUint();

  // Update InfoID / WarningID / ErrorID
  CASE _rspHeader.AlarmMessageSeverity OF

    // Informative message
    Severity.INFO        : InfoID    := _rspHeader.AlarmMessageCode;
    // Warning message
    Severity.WARNING     : WarningID := _rspHeader.AlarmMessageCode;
    // Error message
    Severity.ERROR       : ErrorID   := _rspHeader.AlarmMessageCode;
    // Fataö error message
    Severity.FATAL_ERROR : ErrorID   := _rspHeader.AlarmMessageCode;

  END_CASE

  ParseResponsePayload := ResponseData.PayloadPtr;

END_METHOD

METHOD PROTECTED Reset : DINT
VAR_INPUT
END_VAR

  _uniqueId := 0;
  _stepCmd  := 0;
  Error     := FALSE;
  ErrorID   := 0;
  WarningID := 0;
  InfoID    := 0;

  Reset := RobotLibraryConstants.OK;

END_METHOD

(* ---- RobotLibraryLogFB.st ---- *)
FUNCTION_BLOCK RobotLibraryLogFB
// -------------------------------------------------------------------------
//  SRCI Robot Library
// -------------------------------------------------------------------------
//
//  Object:      RobotLibraryLogFB
//  Author:      Thorsten Brach
//  Date:        2024-11-10
//
//  Description:
//
//
//  Copyright:
//    (C) 2024 Thorsten Brach. All rights reserved
//             Licensed under the LGPL-3.0 license.
//
//  Disclaimer:
//    This project is provided without any guarantee and can be used for
//    private and commercial purposes. Any use is at the user’s
//    own risk and responsibility.
//
// -------------------------------------------------------------------------
VAR_INPUT
  /// Interface to an external logger
  ExternalLogger : IMessageLogger;
  /// Logging level
  LogLevel       : LogLevelEnum := LogLevelEnum.INFO;
END_VAR

VAR
  /// Type of the function block
 _myType         : STRING;
END_VAR

END_FUNCTION_BLOCK

METHOD CreateLogMessage
VAR_INPUT
  /// Timestamp
  Timestamp   : DT;
  /// Type of message according to Table 5-46:
  MessageType : MessageType;
  /// Severity of message according to Table 5-47: Debug, Info, Warning, Error, Fatal error
  Severity    : Severity;
  /// Code of messages
  MessageCode : DWORD;
  /// Static text of message
  MessageText : STRING(255);
END_VAR

VAR
  /// internal log message
 _logMessage : AlarmMessage;
END_VAR

  IF (( ExternalLogger <> 0        ) AND
      ( LogLevel       <= Severity )) {warning 'ToDo: LogLevel and Severity are the same -> use an alias for it'}
  THEN
   _logMessage.Timestamp   := Timestamp;
   _logMessage.MessageType := MessageType;
   _logMessage.Severity    := Severity;
   _logMessage.MessageCode := MessageCode;
   _logMessage.MessageText := StrPadRight(MyType,' ', RobotLibraryDefines.MaxTypeNameLength);
   _logMessage.MessageText := CONCAT(_logMessage.MessageText, ': ');
   _logMessage.MessageText := CONCAT(_logMessage.MessageText,MessageText);

    ExternalLogger.AddMessageLog( _logMessage);
  END_IF

END_METHOD

METHOD CreateLogMessagePara1
VAR_INPUT
  /// Timestamp
  Timestamp   : DT;
  /// Type of message according to Table 5-46:
  MessageType : MessageType;
  /// Severity of message according to Table 5-47: Debug, Info, Warning, Error, Fatal error
  Severity    : Severity;
  /// Code of messages
  MessageCode : DWORD;
  /// Static text of message
  MessageText : STRING(255);
  /// sub string which will replace the placeholder {1}
  Para1       : STRING(255);
END_VAR
VAR
  /// internal log message
 _logMessage : AlarmMessage;
END_VAR

  MessageText := StrReplace(MessageText,'{1}', Para1);

  CreateLogMessage( Timestamp   := Timestamp,
                    MessageType := MessageType,
                    Severity    := Severity,
                    MessageCode := MessageCode,
                    MessageText := MessageText);

END_METHOD

METHOD CreateLogMessagePara2 : BOOL
VAR_INPUT
  /// Timestamp
  Timestamp   : DT;
  /// Type of message according to Table 5-46:
  MessageType : MessageType;
  /// Severity of message according to Table 5-47: Debug, Info, Warning, Error, Fatal error
  Severity    : Severity;
  /// Code of messages
  MessageCode : DWORD;
  /// Static text of message
  MessageText : STRING(255);
  /// sub string which will replace the placeholder {1}
  Para1       : STRING(255);
  /// sub string which will replace the placeholder {2}
  Para2       : STRING(255);
END_VAR
VAR
  /// internal log message
 _logMessage : AlarmMessage;
END_VAR

  MessageText := StrReplace(MessageText,'{2}', Para2);

  CreateLogMessagePara1( Timestamp   := Timestamp,
                         MessageType := MessageType,
                         Severity    := Severity,
                         MessageCode := MessageCode,
                         MessageText := MessageText,
                         Para1       := Para1);

END_METHOD

METHOD CreateLogMessagePara3
VAR_INPUT
  /// Timestamp
  Timestamp   : DT;
  /// Type of message according to Table 5-46:
  MessageType : MessageType;
  /// Severity of message according to Table 5-47: Debug, Info, Warning, Error, Fatal error
  Severity    : Severity;
  /// Code of messages
  MessageCode : DWORD;
  /// Static text of message
  MessageText : STRING(255);
  /// sub string which will replace the placeholder {1}
  Para1       : STRING(255);
  /// sub string which will replace the placeholder {2}
  Para2       : STRING(255);
  /// sub string which will replace the placeholder {3}
  Para3       : STRING(255);
END_VAR
VAR
  /// internal log message
 _logMessage : AlarmMessage;
END_VAR

  MessageText := StrReplace(MessageText,'{3}', Para3);

  CreateLogMessagePara2( Timestamp   := Timestamp,
                         MessageType := MessageType,
                         Severity    := Severity,
                         MessageCode := MessageCode,
                         MessageText := MessageText,
                         Para1       := Para1,
                         Para2       := Para2);

END_METHOD

METHOD CreateLogMessagePara4 : BOOL
VAR_INPUT
  /// Timestamp
  Timestamp   : DT;
  /// Type of message according to Table 5-46:
  MessageType : MessageType;
  /// Severity of message according to Table 5-47: Debug, Info, Warning, Error, Fatal error
  Severity    : Severity;
  /// Code of messages
  MessageCode : DWORD;
  /// Static text of message
  MessageText : STRING(255);
  /// sub string which will replace the placeholder {1}
  Para1       : STRING(255);
  /// sub string which will replace the placeholder {2}
  Para2       : STRING(255);
  /// sub string which will replace the placeholder {3}
  Para3       : STRING(255);
  /// sub string which will replace the placeholder {4}
  Para4       : STRING(255);
END_VAR
VAR
  /// internal log message
 _logMessage : AlarmMessage;
END_VAR

  MessageText := StrReplace(MessageText,'{4}', Para4);

  CreateLogMessagePara3( Timestamp   := Timestamp,
                         MessageType := MessageType,
                         Severity    := Severity,
                         MessageCode := MessageCode,
                         MessageText := MessageText,
                         Para1       := Para1,
                         Para2       := Para2,
                         Para3       := Para3);

END_METHOD

METHOD CreateLogMessagePara5
VAR_INPUT
  /// Timestamp
  Timestamp   : DT;
  /// Type of message according to Table 5-46:
  MessageType : MessageType;
  /// Severity of message according to Table 5-47: Debug, Info, Warning, Error, Fatal error
  Severity    : Severity;
  /// Code of messages
  MessageCode : DWORD;
  /// Static text of message
  MessageText : STRING(255);
  /// sub string which will replace the placeholder {1}
  Para1       : STRING(255);
  /// sub string which will replace the placeholder {2}
  Para2       : STRING(255);
  /// sub string which will replace the placeholder {3}
  Para3       : STRING(255);
  /// sub string which will replace the placeholder {4}
  Para4       : STRING(255);
  /// sub string which will replace the placeholder {5}
  Para5       : STRING(255);
END_VAR
VAR
  /// internal log message
 _logMessage : AlarmMessage;
END_VAR

  MessageText := StrReplace(MessageText,'{5}', Para5);

  CreateLogMessagePara4( Timestamp   := Timestamp,
                         MessageType := MessageType,
                         Severity    := Severity,
                         MessageCode := MessageCode,
                         MessageText := MessageText,
                         Para1       := Para1,
                         Para2       := Para2,
                         Para3       := Para3,
                         Para4       := Para4);

END_METHOD

PROPERTY PROTECTED MyType : STRING

GET
VAR
END_VAR

  MyType := _myType;

END_GET

SET
VAR
END_VAR

  _myType := MyType;

  // set the max type name length
  RobotLibraryDefines.MaxTypeNameLength := MAX(LEN(_myType), RobotLibraryDefines.MaxTypeNameLength);

END_SET

(* ---- SendData.st ---- *)
{attribute 'pack_mode' := '1'}
FUNCTION_BLOCK SendData
// -------------------------------------------------------------------------
//  SRCI Robot Library
// -------------------------------------------------------------------------
//
//  Object:      SendData
//  Author:      Thorsten Brach
//  Date:        2024-06-01
//
//  Description:
//
//
//  Copyright:
//    (C) 2024 Thorsten Brach. All rights reserved
//             Licensed under the LGPL-3.0 license.
//
//  Disclaimer:
//    This project is provided without any guarantee and can be used for
//    private and commercial purposes. Any use is at the user’s
//    own risk and responsibility.
//
// -------------------------------------------------------------------------
VAR_INPUT
  /// Payload
  Payload    : ARRAY [0..RobotLibraryParameter.TELEGRAM_PAYLOAD_MAX] OF BYTE;
  /// Payload length
  PayloadLen : UDINT;
  /// Payload pointer
  PayloadPtr : UDINT;
END_VAR

END_FUNCTION_BLOCK

/// Adds a ArmConfigParameter to the payload buffer, increase the payload pointer and returns the payload lenght
METHOD AddArmConfig : UDINT
VAR_INPUT
  /// Value to add
  Value : ArmConfigParameter;
END_VAR

VAR
  /// temporary Byte
 _tmpByte : BYTE;
END_VAR

  Value := Value;

  _tmpByte.0 := Value.Shoulder = ArmConfigShoulder.USE_CONFIG;
  _tmpByte.1 := Value.Elbow    = ArmConfigElbow   .USE_CONFIG;
  _tmpByte.2 := Value.Wrist    = ArmConfigWrist   .USE_CONFIG;

  AddByte(_tmpByte);
  AddByte(0);

  AddArmConfig := PayloadLen;

END_METHOD

/// Adds a BOOL to the payload buffer, increase the payload pointer and returns the payload lenght
METHOD AddBool : UDINT
VAR_INPUT
  /// Value to add
  Value : BOOL;
END_VAR

VAR
  /// temporary byte
 _tmpByte : BYTE := 0;
END_VAR

  _tmpByte.0 := Value;
  // copy data
  MemCpy( ADR(Payload[PayloadPtr]), ADR(_tmpByte), SIZEOF(_tmpByte));
  // inc payload pointer
  PayloadPtr := PayloadPtr + SIZEOF(_tmpByte);
  // return payload len
  AddBool := PayloadLen := PayloadPtr;

END_METHOD

/// Adds a BYTE to the payload buffer, increase the payload pointer and returns the payload lenght
METHOD AddByte : UDINT
VAR_INPUT
  /// Value to add
  Value : BYTE;
END_VAR

  Value := Value;
  // copy data
  MemCpy( ADR(Payload[PayloadPtr]), ADR(Value), SIZEOF(Value));
  // inc payload pointer
  PayloadPtr := PayloadPtr + SIZEOF(Value);
  // return payload len
  AddByte := PayloadLen := PayloadPtr;

END_METHOD

/// Adds a DataBlock to the payload buffer, increase the payload pointer and returns the payload lenght
METHOD AddDataBlock : UDINT
VAR_INPUT
  /// Value to add
  pValue : POINTER TO BYTE;
  /// Size of data block
  Size   : UDINT;
END_VAR

  IF (pValue = 0) OR (Size = 0 )
  THEN
    RETURN;
  END_IF

  // copy data
  MemCpy( ADR(Payload[PayloadPtr]), pValue, Size);
  // inc payload pointer
  PayloadPtr := PayloadPtr + Size;
  // return payload len
  AddDataBlock := PayloadLen := PayloadPtr;

END_METHOD

/// Adds a DataInSync to the payload buffer, increase the payload pointer and returns the payload lenght
METHOD AddDataEnableSync : UDINT
VAR_INPUT
  /// Value to add
  Value : DataEnableSync;
END_VAR

VAR
  /// temporary Byte
 _tmpByte : BYTE;
END_VAR

  Value := Value;

  _tmpByte.0 := Value.EnableSyncTool;
  _tmpByte.1 := Value.EnableSyncFrame;
  _tmpByte.2 := Value.EnableSyncLoad;
  _tmpByte.3 := Value.EnableSyncWorkArea;
  _tmpByte.4 := Value.EnableSyncSWLimits;
  _tmpByte.5 := Value.EnableSyncDefaultDynamics;
  _tmpByte.5 := Value.EnableSyncReferenceDynamics;
  _tmpByte.6 := Value.AllowDynamicBlending;

  AddByte(_tmpByte);

  AddDataEnableSync := PayloadLen;

END_METHOD

/// Adds a DataInSync to the payload buffer, increase the payload pointer and returns the payload lenght
METHOD AddDataInSync : UDINT
VAR_INPUT
  /// Value to add
  Value : DataInSync;
END_VAR

VAR
  /// temporary Byte
 _tmpByte : BYTE;
END_VAR

  Value := Value;

  _tmpByte.0 := Value.ToolsInSync;
  _tmpByte.1 := Value.FramesInSync;
  _tmpByte.2 := Value.LoadsInSync;
  _tmpByte.3 := Value.WorkAreasInSync;
  _tmpByte.4 := Value.SoftwareLimitsInSync;
  _tmpByte.5 := Value.DefaultDynamicsInSync;
  _tmpByte.5 := Value.ReferenceDynamicsInSync;

  AddByte(_tmpByte);

  AddDataInSync := PayloadLen;

END_METHOD

/// Adds a DWORD to the payload buffer , increase the payload pointer and returns the payload lenght
METHOD AddDword : UDINT
VAR_INPUT
  /// Value to add
  Value : DWORD;
END_VAR

  // swap byte order
  Value := SwapDword(Value);
  // copy data
  MemCpy( ADR(Payload[PayloadPtr]), ADR(Value), SIZEOF(Value));
  // inc data index
  PayloadPtr := PayloadPtr + SIZEOF(Value);
  // return payload len
  AddDword := PayloadLen := PayloadPtr;

END_METHOD

/// Adds two halfe BYTE to the payload buffer , increase the payload pointer and returns the payload lenght
METHOD AddHalfBytes : UDINT
VAR_INPUT
  /// Value to add
  HalfByteHi : BYTE;
  /// Value to add
  HalfByteLo : BYTE;
END_VAR

VAR
  /// internal value
 _value : BYTE;
END_VAR

  _value := CombineHalfBytes( HalfByteHi := HalfByteHi, HalfByteLo := HalfByteLo);
  // copy data
  MemCpy( ADR(Payload[PayloadPtr]), ADR(_value), SIZEOF(_value));
  // inc payload pointer
  PayloadPtr := PayloadPtr + SIZEOF(_value);
  // return payload len
  AddHalfBytes := PayloadLen := PayloadPtr;

END_METHOD

/// Adds a IEC_DATE to the payload buffer, increase the payload pointer and returns the payload lenght
METHOD AddIecDate : UDINT
VAR_INPUT
  /// Value to add
  Value : IEC_DATE;
END_VAR

  Value := SwapIecDate(Value);
  // copy data
  MemCpy( ADR(Payload[PayloadPtr]), ADR(Value), SIZEOF(Value));
  // inc payload pointer
  PayloadPtr := PayloadPtr + SIZEOF(Value);
  // return payload len
  AddIecDate := PayloadLen := PayloadPtr;

END_METHOD

/// Adds a IEC_TIME to the payload buffer, increase the payload pointer and returns the payload lenght
METHOD AddIecTime : UDINT
VAR_INPUT
  /// Value to add
  Value : IEC_TIME;
END_VAR

  Value := SwapIecTime(Value);
  // copy data
  MemCpy( ADR(Payload[PayloadPtr]), ADR(Value), SIZEOF(Value));
  // inc payload pointer
  PayloadPtr := PayloadPtr + SIZEOF(Value);
  // return payload len
  AddIecTime := PayloadLen := PayloadPtr;

END_METHOD

/// Adds a INT to the payload buffer , increase the payload pointer and returns the payload lenght
METHOD AddInt : UDINT
VAR_INPUT
  /// Value to add
  Value : INT;
END_VAR

  // swap byte order
  Value := SwapInt(Value);
  // copy data
  MemCpy( ADR(Payload[PayloadPtr]), ADR(Value), SIZEOF(Value));
  // inc data index
  PayloadPtr := PayloadPtr + SIZEOF(Value);
  // return payload len
  AddInt := PayloadLen := PayloadPtr;

END_METHOD

/// Adds a REAL to the payload buffer , increase the payload pointer and returns the payload lenght
METHOD AddReal : UDINT
VAR_INPUT
  /// Value to add
  Value : REAL;
END_VAR

  // swap byte order
  Value := SwapReal(Value);
  // copy data
  MemCpy( ADR(Payload[PayloadPtr]), ADR(Value), SIZEOF(Value));
  // inc data index
  PayloadPtr := PayloadPtr + SIZEOF(Value);
  // return payload len
  AddReal := PayloadLen := PayloadPtr;

END_METHOD

/// Adds a SINT to the payload buffer, increase the payload pointer and returns the payload lenght
METHOD AddSint : UDINT
VAR_INPUT
  /// Value to add
  Value : SINT;
END_VAR

  Value := Value;
  // copy data
  MemCpy( ADR(Payload[PayloadPtr]), ADR(Value), SIZEOF(Value));
  // inc payload pointer
  PayloadPtr := PayloadPtr + SIZEOF(Value);
  // return payload len
  AddSint := PayloadLen := PayloadPtr;

END_METHOD

/// Adds a String to the payload buffer, increase the payload pointer and returns the payload lenght
METHOD AddString : UDINT
VAR_INPUT
  /// Value to add
  Value : STRING(255);
END_VAR

  IF ( LEN(Value) = 0 )
  THEN
    RETURN;
  END_IF

  // copy data
  MemCpy( ADR(Payload[PayloadPtr]), ADR(Value), DINT_TO_UDINT(LEN(Value)));
  // inc payload pointer
  PayloadPtr := PayloadPtr + DINT_TO_UDINT(LEN(Value));
  // return payload len
  AddString := PayloadLen := PayloadPtr;

END_METHOD

/// Adds a TIME to the payload buffer , increase the payload pointer and returns the payload lenght
METHOD AddTime : UDINT
VAR_INPUT
  /// Value to add
  Value : TOD;
END_VAR

  // swap byte order
  Value := SwapIecTime(Value);
  // copy data
  MemCpy( ADR(Payload[PayloadPtr]), ADR(Value), SIZEOF(Value));
  // inc data index
  PayloadPtr := PayloadPtr + SIZEOF(Value);
  // return payload len
  AddTime := PayloadLen := PayloadPtr;

END_METHOD

/// Adds a TurnNumber to the payload buffer, increase the payload pointer and returns the payload lenght
METHOD AddTurnNumber : UDINT
VAR_INPUT
  /// Value to add
  Value : TurnNumber;
END_VAR

VAR
  /// temporary Byte
 _tmpByte : BYTE;
END_VAR

  Value := Value;

  AddHalfBytes( HalfByteHi := SINT_TO_BYTE(Value.J2Turns) , HalfByteLo := SINT_TO_BYTE(Value.J1Turns));
  AddHalfBytes( HalfByteHi := SINT_TO_BYTE(Value.J4Turns) , HalfByteLo := SINT_TO_BYTE(Value.J3Turns));
  AddHalfBytes( HalfByteHi := SINT_TO_BYTE(Value.J6Turns) , HalfByteLo := SINT_TO_BYTE(Value.J5Turns));
  AddByte(SINT_TO_BYTE(Value.E1Turns));

  AddTurnNumber := PayloadLen;

END_METHOD

/// Adds a UDINT to the payload buffer , increase the payload pointer and returns the payload lenght
METHOD AddUdint : UDINT
VAR_INPUT
  /// Value to add
  Value : UDINT;
END_VAR

  // swap byte order
  Value := SwapUdint(Value);
  // copy data
  MemCpy( ADR(Payload[PayloadPtr]), ADR(Value), SIZEOF(Value));
  // inc data index
  PayloadPtr := PayloadPtr + SIZEOF(Value);
  // return payload len
  AddUdint := PayloadLen := PayloadPtr;

END_METHOD

/// Adds a UINT to the payload buffer , increase the payload pointer and returns the payload lenght
METHOD AddUint : UDINT
VAR_INPUT
  /// Value to add
  Value : UINT;
END_VAR

  // swap byte order
  Value := SwapUint(Value);
  // copy data
  MemCpy( ADR(Payload[PayloadPtr]), ADR(Value), SIZEOF(Value));
  // inc data index
  PayloadPtr := PayloadPtr + SIZEOF(Value);
  // return payload len
  AddUint := PayloadLen := PayloadPtr;

END_METHOD

/// Adds a USINT to the payload buffer, increase the payload pointer and returns the payload lenght
METHOD AddUsint : UDINT
VAR_INPUT
  /// Value to add
  Value : USINT;
END_VAR

  Value := Value;
  // copy data
  MemCpy( ADR(Payload[PayloadPtr]), ADR(Value), SIZEOF(Value));
  // inc payload pointer
  PayloadPtr := PayloadPtr + SIZEOF(Value);
  // return payload len
  AddUsint := PayloadLen := PayloadPtr;

END_METHOD

/// Resets the payload buffer, the payload pointer and the payload length
METHOD Reset
VAR_INPUT
END_VAR

  MemSet(ADR(Payload), 0 , SIZEOF(Payload));
  PayloadLen := 0;
  PayloadPtr := 0;

END_METHOD
